FUNCTION_BLOCK FB_CondensingBoiler EXTENDS FB_ActuatorContinous
VAR_INPUT
END_VAR
VAR_OUTPUT
	bError : BOOL;
END_VAR
VAR
	{attribute 'OPC.UA.DA' := '1'}
	localState : ST_CondensingBoilerState;
	
	//default parameters
	localDefaultParameters : ST_CondensingBoilerDefaultParameters;
	
	//analog converters
	OutputConverter : FB_AnalogOutput(fUpperLimit := 100, fLowerLimit := 0);
	
	//I/O Links
	nSetPoint_OUT			AT %Q* : INT;
	bSetStatusOn_OUT 		AT %Q* : BOOL;
	bStatusOn_IN			AT %I* : BOOL;
	bError_IN 				AT %I* : BOOL;
END_VAR

MAIN();
OutputConverter(fValue := fSetPoint);

METHOD GetState : BOOL
VAR_INPUT
END_VAR
//local state
controlState.bStatusOn := bStatusOn_IN;
localState.bError := bError_IN;
bStatusOn := controlState.bStatusOn;
bError := localState.bError;
END_METHOD

METHOD PROTECTED  SetSetPointLimits : BOOL
VAR_INPUT
END_VAR
aSetPointLimits[1] := localDefaultParameters.aSetPointLimitsTemperature[1];
aSetPointLimits[2] := localDefaultParameters.aSetPointLimitsTemperature[2];
END_METHOD

METHOD SetState : BOOL
VAR_INPUT
END_VAR
setPointState.fSetPoint := fSetPoint;
setPointState.aSetPointLimits := aSetPointLimits;
setPointState.sSetPointUnit := 'degreeC';

nSetPoint_OUT := OutputConverter.nValue;  //converts real setpoint for terminal
bSetStatusOn_OUT := bSetStatusOn;
END_METHOD

PROPERTY ST_DefaultParameters : REFERENCE TO ST_CondensingBoilerDefaultParameters
GET
ST_DefaultParameters REF= localDefaultParameters;
END_GET
SET
localDefaultParameters := ST_DefaultParameters;
END_SET
END_PROPERTY

END_FUNCTION_BLOCK

(* stored: Version 1.1.0.1, ProductVersion 3.1.4024.10
   POU FB_CondensingBoiler: Id {532a516d-9cc8-4820-b59b-bc9ad3e263f3}, SpecialFunc None
   Method GetState: Id {a0e81b08-f1df-4174-9a0b-7e03b77586a6}
   Method SetSetPointLimits: Id {ae6e5319-fa8e-4a57-953e-0d088040aef7}
   Method SetState: Id {3868a82c-54c5-4a4b-a783-f9cc61cf38bb}
   Property ST_DefaultParameters: Id {4e5c1c85-1fd7-4ebd-bb6e-1f11f763d57a}
   Get Get: Id {3713ad30-46db-4a2e-87f1-58aab8856e42}
   Set Set: Id {19f4adf1-6b65-4425-87a1-833a085f1d8b} *)
